FUNCTION_BLOCK Q_ESC_AX (* Esc Command with AX adapter ( Part 6 - F.8 ) *)
  (* Standard: ISO 11783-6; Description: Copyright (c) 2026 Meisterschulen am Ostbahnhof This program and the accompanying materials are made available under the terms of the Eclipse Public License 2.0 which is available at https://www.eclipse.org/legal/epl-2.0/ SPDX-License-Identifier: EPL-2.0 *)
  (* Version 1.0, 2026-09-11, Franz Höpfinger, Meisterschulen am Ostbahnhof, AX adapter wrapper for Q_ESC *)
  PACKAGE isobus::UT::Q;
  (* Documentation:
  Esc Command with AX adapter ( Part 6 - F.8 )
   This FB is an AX adapter wrapper around Q_ESC.
  *)
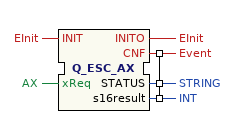
  EVENT_INPUT
    INIT : EInit; (* Service Initialization *)
  END_EVENT
  EVENT_OUTPUT
    INITO : EInit; (* Initialization Confirm *)
    CNF WITH STATUS, s16result; (* Confirmation of Requested Service *)
  END_EVENT
  VAR_OUTPUT
    STATUS : STRING; (* Service Status *)
    s16result : INT; (* retval see description *)
  END_VAR
  SOCKETS
    xReq : adapter::types::unidirectional::AX; (* Esc Command Trigger *)
  END_SOCKETS
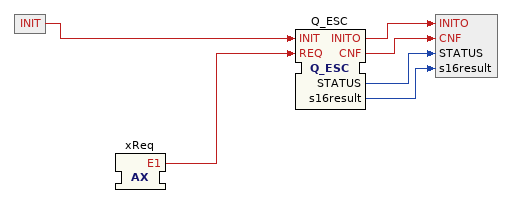
  FBS
    Q_ESC : isobus::UT::Q::Q_ESC;
  END_FBS
  EVENT_CONNECTIONS
    INIT TO Q_ESC.INIT;
    Q_ESC.INITO TO INITO;
    Q_ESC.CNF TO CNF;
    xReq.E1 TO Q_ESC.REQ;
  END_CONNECTIONS
  DATA_CONNECTIONS
    Q_ESC.STATUS TO STATUS;
    Q_ESC.s16result TO s16result;
  END_CONNECTIONS
END_FUNCTION_BLOCK
